ABB RobotStudio station: 501_cocktailBot_v1_20220412-142528.rsstn

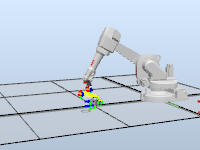
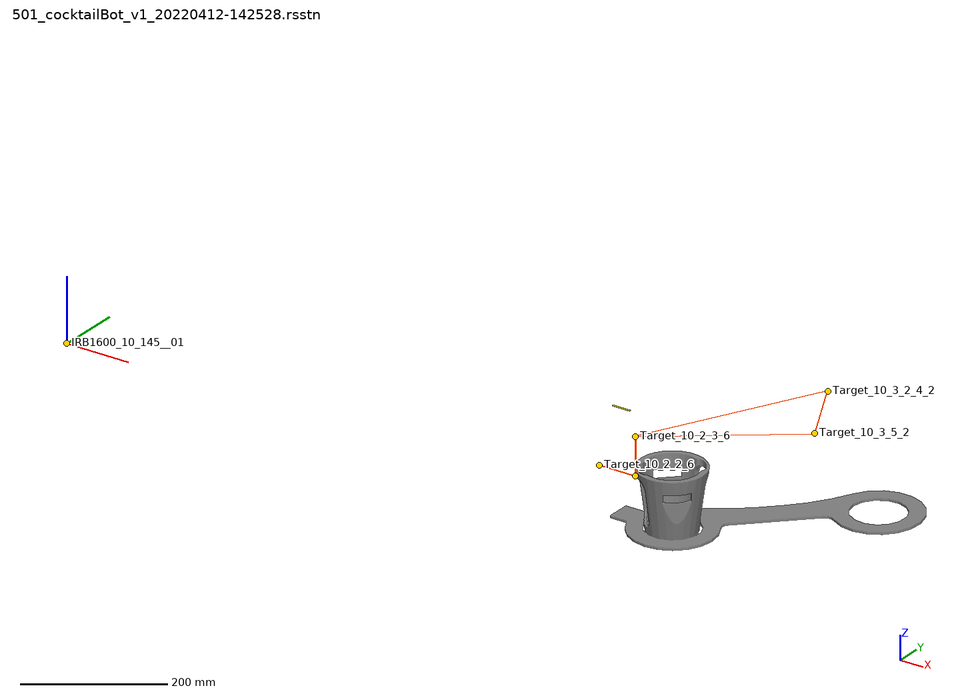
[picture v1: parts stored in the station drawn from their meshes, with robot base, taught points and paths (robot models come from the ABB library and are not in the file)]
Station 501_cocktailBot_v1 (saved by RobotStudio 21.4.9700.0)
Controller IRB1600_10_145
  mechanical unit ROB_1: IRB1600_10_145__01, 6 joints, base frame (0, 0, 0) mm
Layout (positions relative to the parent item):
  - GS25_Gripper [mechanism] at (1000, -191.15, 290.13) mm, rotated rx -130 ry 0 rz 0 deg; joint values [0, 0] (rad or m)
      TCP GS25_Gripper_1 at (0, 0, 90.5) mm
      links: L1, L2, L3
  - Gripper_SC [smart component] at (990, 0, 0) mm, rotated rx 0 ry 90 rz 0 deg
      signals: DI Gripper_Attach, DO Attached
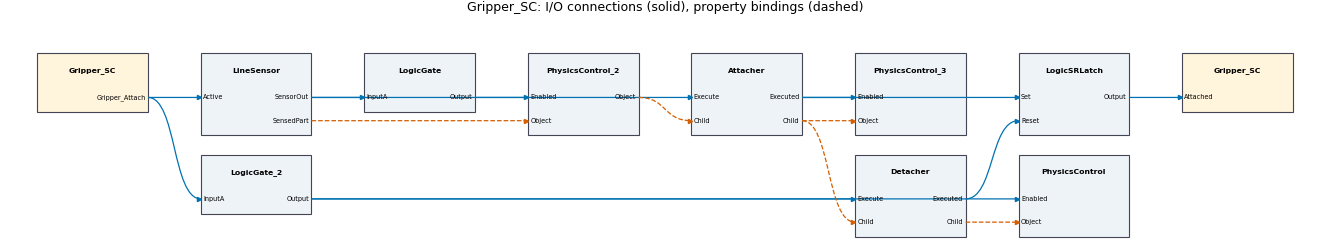
      connections:
        Gripper_SC.Gripper_Attach -> LineSensor.Active
        LineSensor.SensorOut -> LogicGate.InputA
        LogicGate.Output -> PhysicsControl_2.Enabled
        LineSensor.SensorOut -> Attacher.Execute
        Attacher.Executed -> LogicSRLatch.Set
        LogicSRLatch.Output -> Gripper_SC.Attached
        Gripper_SC.Gripper_Attach -> LogicGate_2.InputA
        LogicGate_2.Output -> Detacher.Execute
        Detacher.Executed -> LogicSRLatch.Reset
        LogicGate_2.Output -> PhysicsControl.Enabled
        Attacher.Executed -> PhysicsControl_3.Enabled
        LineSensor.SensedPart => PhysicsControl_2.Object
        PhysicsControl_2.Object => Attacher.Child
        Detacher.Child => PhysicsControl.Object
        Attacher.Child => Detacher.Child
        Attacher.Child => PhysicsControl_3.Object
    - LineSensor [smart component, from Components\LineSensor.rslib] at (-231.47, -121.24, -10.63) mm, rotated rx 0 ry 0 rz 50 deg
        properties: Start=[2.85358248322543E-07 0 0.00610500428453198]; End=[2.85358248322543E-07 0 0.0350726372106779]; Radius=0.001; SensedPart=(none); SensedPoint=[0 0 0]
      - _sensorPart_ [part], size 2 x 2 x 29 mm
    - Attacher [smart component, from Components\Attacher.rslib]
        properties: Parent=GS25_Gripper; Flange=0; Child=cup; Mount=false; Offset=[0 0 0]; Orientation=[0 0 0]
    - Detacher [smart component, from Components\Detacher.rslib]
        properties: Child=cup; KeepPosition=true
    - LogicGate [smart component, from Components\LogicGate.rslib]
        properties: Operator=NOT; Delay=0
    - LogicSRLatch [smart component, from Components\LogicSRLatch.rslib]
    - PhysicsControl [smart component, from Components\PhysicsControl.rslib]
        properties: Object=cup; Behavior=0; SurfaceVelocity=0
    - LogicGate_2 [smart component, from Components\LogicGate.rslib]
        properties: Operator=NOT; Delay=0
    - PhysicsControl_2 [smart component, from Components\PhysicsControl.rslib]
        properties: Object=(none); Behavior=3; SurfaceVelocity=0
  - SmartComponent_1 [smart component] at (1000, -121.83, 231.96) mm, rotated rx -130 ry 0 rz 0 deg
      signals: DI Reset_cube, DI Reset_objects
      connections:
        SmartComponent_1.Reset_objects -> Positioner.Execute
        Positioner.Executed -> Positioner_2.Execute
        Positioner_2.Executed -> Positioner_3.Execute
    - Positioner [smart component, from Components\Positioner.rslib]
        properties: Object=(none); Position=[-0.449454 -0.908727 0]; Orientation=[1.5707963267949 0 1.5707963267949]; Reference=Global; ReferenceObject=(none)
    - Positioner_2 [smart component, from Components\Positioner.rslib]
        properties: Object=(none); Position=[-0.498778 -0.908734 0.000796]; Orientation=[1.5707963267949 0 -1.56573487196411]; Reference=Global; ReferenceObject=(none)
    - Positioner_3 [smart component, from Components\Positioner.rslib]
        properties: Object=(none); Position=[-0.452858 -1.056064 0.000796]; Orientation=[1.5707963267949 0 -1.37980494674916]; Reference=Global; ReferenceObject=(none)
  - Toolside_plates [part] at (0, 0, 0) mm
  - Toolplate2 [part, from Libraries\gs25V2.rslib] at (0, 0, 0) mm
  - cup [part] at (1000, -1.82, 0) mm, rotated rx 90 ry 0 rz 0 deg, size 101.6 x 95 x 100.9 mm
  - cupHolderHolder_3 [part] at (1000, 0, -1.59) mm, rotated rx -90 ry 0 rz 0 deg, size 355.2 x 3.2 x 329.2 mm
  - IRB1600_10_145__01 [mechanism, from Robots\IRB1600_10_145_G_01.rslib] at (0, 0, 0) mm; joint values [-0.2364, 1.0092, 0.0645, 1.0133, 1.0708, 2.1274] (rad or m)
Attachment: LineSensor is attached to GS25_Gripper / L1
Attachment: SmartComponent_1 is attached to GS25_Gripper / L1
Attachment: GS25_Gripper is attached to IRB1600_10_145__01 / Link6
EventTableEntry 1061: Group=, Trigger=DO_Gripper 1062, Actions=[EventTableActionMechanicalPose 1063], Comment=, ActivationMode=2, Cyclic=false
EventTableTriggerIO 1062: IOValue=[1], IRC5Controller=? -1, Operator=0, SignalSource=? -1
EventTableActionMechanicalPose 1063: VirtualSignal=, Mechanism=GS25_Gripper 1072, ToPoseName=Gripper_Open, VirtualSignalValue=[1]
EventTableEntry 1064: Group=, Trigger=DO_Gripper 1065, Actions=[EventTableActionMechanicalPose 1066], Comment=, ActivationMode=2, Cyclic=false
EventTableTriggerIO 1065: IOValue=[0], IRC5Controller=? -1, Operator=0, SignalSource=? -1
EventTableActionMechanicalPose 1066: VirtualSignal=, Mechanism=GS25_Gripper 1072, ToPoseName=Gripper_Closed, VirtualSignalValue=[1]
EventTableTriggerIO 1240: IOValue=[1], IRC5Controller=? -1, Operator=0, SignalSource=? -1
EventTableTriggerIO 1241: IOValue=[0], IRC5Controller=? -1, Operator=0, SignalSource=? -1
EventTableTriggerIO 1347: IOValue=[1], IRC5Controller=? -1, Operator=0, SignalSource=? -1
EventTableTriggerIO 1348: IOValue=[1], IRC5Controller=? -1, Operator=0, SignalSource=? -1
EventTableTriggerIO 1349: IOValue=[1], IRC5Controller=? -1, Operator=0, SignalSource=? -1
EventTableTriggerIO 1350: IOValue=[1], IRC5Controller=? -1, Operator=0, SignalSource=? -1
EventTableTriggerIO 1351: IOValue=[1], IRC5Controller=? -1, Operator=0, SignalSource=? -1
EventTableTriggerIO 1352: IOValue=[1], IRC5Controller=? -1, Operator=0, SignalSource=? -1
EventTableTriggerIO 1353: IOValue=[0], IRC5Controller=? -1, Operator=0, SignalSource=? -1
EventTableTriggerIO 1354: IOValue=[0], IRC5Controller=? -1, Operator=0, SignalSource=? -1
EventTableTriggerIO 1355: IOValue=[0], IRC5Controller=? -1, Operator=0, SignalSource=? -1
EventTableTriggerIO 1356: IOValue=[0], IRC5Controller=? -1, Operator=0, SignalSource=? -1
EventTableTriggerIO 1357: IOValue=[0], IRC5Controller=? -1, Operator=0, SignalSource=? -1
EventTableTriggerIO 1358: IOValue=[0], IRC5Controller=? -1, Operator=0, SignalSource=? -1
EventTableTriggerIO 1359: IOValue=[1], IRC5Controller=? -1, Operator=0, SignalSource=? -1
EventTableTriggerIO 1360: IOValue=[0], IRC5Controller=? -1, Operator=0, SignalSource=? -1
EventTableTriggerIO 2021: IOValue=[1], IRC5Controller=? -1, Operator=0, SignalSource=? -1
EventTableTriggerIO 2022: IOValue=[0], IRC5Controller=? -1, Operator=0, SignalSource=? -1
EventTableTriggerIO 2984: IOValue=[1], IRC5Controller=? -1, Operator=0, SignalSource=? -1
EventTableTriggerIO 2985: IOValue=[1], IRC5Controller=? -1, Operator=0, SignalSource=? -1
EventTableTriggerIO 2986: IOValue=[1], IRC5Controller=? -1, Operator=0, SignalSource=? -1
EventTableTriggerIO 2987: IOValue=[1], IRC5Controller=? -1, Operator=0, SignalSource=? -1
EventTableTriggerIO 2988: IOValue=[1], IRC5Controller=? -1, Operator=0, SignalSource=? -1
EventTableTriggerIO 2989: IOValue=[1], IRC5Controller=? -1, Operator=0, SignalSource=? -1
EventTableTriggerIO 2990: IOValue=[0], IRC5Controller=? -1, Operator=0, SignalSource=? -1
EventTableTriggerIO 2991: IOValue=[0], IRC5Controller=? -1, Operator=0, SignalSource=? -1
EventTableTriggerIO 2992: IOValue=[0], IRC5Controller=? -1, Operator=0, SignalSource=? -1
EventTableTriggerIO 2993: IOValue=[0], IRC5Controller=? -1, Operator=0, SignalSource=? -1
EventTableTriggerIO 2994: IOValue=[0], IRC5Controller=? -1, Operator=0, SignalSource=? -1
EventTableTriggerIO 2995: IOValue=[0], IRC5Controller=? -1, Operator=0, SignalSource=? -1
EventTableTriggerIO 3347: IOValue=[1], IRC5Controller=? -1, Operator=0, SignalSource=? -1
EventTableTriggerIO 3348: IOValue=[0], IRC5Controller=? -1, Operator=0, SignalSource=? -1
EventTableTriggerIO 3367: IOValue=[1], IRC5Controller=? -1, Operator=0, SignalSource=? -1
EventTableTriggerIO 3368: IOValue=[1], IRC5Controller=? -1, Operator=0, SignalSource=? -1
EventTableTriggerIO 3369: IOValue=[1], IRC5Controller=? -1, Operator=0, SignalSource=? -1
EventTableTriggerIO 3370: IOValue=[1], IRC5Controller=? -1, Operator=0, SignalSource=? -1
EventTableTriggerIO 3371: IOValue=[1], IRC5Controller=? -1, Operator=0, SignalSource=? -1
EventTableTriggerIO 3372: IOValue=[1], IRC5Controller=? -1, Operator=0, SignalSource=? -1
EventTableTriggerIO 3373: IOValue=[1], IRC5Controller=? -1, Operator=0, SignalSource=? -1
EventTableTriggerIO 3374: IOValue=[1], IRC5Controller=? -1, Operator=0, SignalSource=? -1
EventTableTriggerIO 3375: IOValue=[1], IRC5Controller=? -1, Operator=0, SignalSource=? -1
EventTableTriggerIO 3376: IOValue=[1], IRC5Controller=? -1, Operator=0, SignalSource=? -1
EventTableTriggerIO 3377: IOValue=[1], IRC5Controller=? -1, Operator=0, SignalSource=? -1
EventTableTriggerIO 3378: IOValue=[0], IRC5Controller=? -1, Operator=0, SignalSource=? -1
EventTableTriggerIO 3379: IOValue=[0], IRC5Controller=? -1, Operator=0, SignalSource=? -1
EventTableTriggerIO 3380: IOValue=[0], IRC5Controller=? -1, Operator=0, SignalSource=? -1
EventTableTriggerIO 3381: IOValue=[0], IRC5Controller=? -1, Operator=0, SignalSource=? -1
EventTableTriggerIO 3382: IOValue=[0], IRC5Controller=? -1, Operator=0, SignalSource=? -1
EventTableTriggerIO 3383: IOValue=[0], IRC5Controller=? -1, Operator=0, SignalSource=? -1
EventTableTriggerIO 3384: IOValue=[0], IRC5Controller=? -1, Operator=0, SignalSource=? -1
EventTableTriggerIO 3385: IOValue=[0], IRC5Controller=? -1, Operator=0, SignalSource=? -1
EventTableTriggerIO 3386: IOValue=[0], IRC5Controller=? -1, Operator=0, SignalSource=? -1
EventTableTriggerIO 3387: IOValue=[0], IRC5Controller=? -1, Operator=0, SignalSource=? -1
EventTableTriggerIO 3388: IOValue=[0], IRC5Controller=? -1, Operator=0, SignalSource=? -1
EventTableTriggerIO 3593: IOValue=[1], IRC5Controller=? -1, Operator=0, SignalSource=? -1
EventTableTriggerIO 3594: IOValue=[1], IRC5Controller=? -1, Operator=0, SignalSource=? -1
EventTableTriggerIO 3595: IOValue=[1], IRC5Controller=? -1, Operator=0, SignalSource=? -1
EventTableTriggerIO 3596: IOValue=[1], IRC5Controller=? -1, Operator=0, SignalSource=? -1
EventTableTriggerIO 3597: IOValue=[0], IRC5Controller=? -1, Operator=0, SignalSource=? -1
EventTableTriggerIO 3598: IOValue=[0], IRC5Controller=? -1, Operator=0, SignalSource=? -1
EventTableTriggerIO 3599: IOValue=[0], IRC5Controller=? -1, Operator=0, SignalSource=? -1
EventTableTriggerIO 3600: IOValue=[0], IRC5Controller=? -1, Operator=0, SignalSource=? -1
EventTableTriggerIO 3620: IOValue=[1], IRC5Controller=? -1, Operator=0, SignalSource=? -1
EventTableTriggerIO 3621: IOValue=[0], IRC5Controller=? -1, Operator=0, SignalSource=? -1
EventTableTriggerIO 3624: IOValue=[1], IRC5Controller=? -1, Operator=0, SignalSource=? -1
EventTableTriggerIO 3625: IOValue=[1], IRC5Controller=? -1, Operator=0, SignalSource=? -1
EventTableTriggerIO 3626: IOValue=[1], IRC5Controller=? -1, Operator=0, SignalSource=? -1
EventTableTriggerIO 3627: IOValue=[0], IRC5Controller=? -1, Operator=0, SignalSource=? -1
EventTableTriggerIO 3628: IOValue=[0], IRC5Controller=? -1, Operator=0, SignalSource=? -1
EventTableTriggerIO 3629: IOValue=[0], IRC5Controller=? -1, Operator=0, SignalSource=? -1
EventTableTriggerIO 3630: IOValue=[1], IRC5Controller=? -1, Operator=0, SignalSource=? -1
EventTableTriggerIO 3631: IOValue=[0], IRC5Controller=? -1, Operator=0, SignalSource=? -1
EventTableTriggerIO 4343: IOValue=[1], IRC5Controller=? -1, Operator=0, SignalSource=? -1
EventTableTriggerIO 4344: IOValue=[0], IRC5Controller=? -1, Operator=0, SignalSource=? -1
Station logic (signal -> signal, property => property):
  IRB_1600_8kg_1.45m.DO_Attach_me -> Gripper_SC.Gripper_Attach
  IRB_1600_8kg_1.45m.DO_Reset_blocks -> SmartComponent_1.Reset_objects
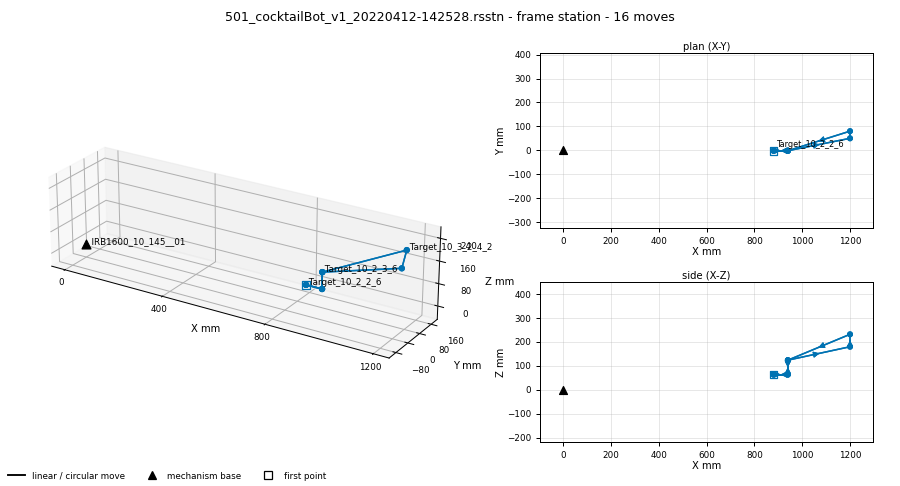
[picture p0: tool path of 501_cocktailBot_v1_20220412-142528.rsstn in frame station, 16 of 17 moves have a stored position in this frame; points joined in program order, loops and branches not executed]
Targets, tools, work objects and paths stored in the station, written as RAPID:
! task (no controller)
MODULE CalibData
  PERS tooldata GS25_Gripper_TCP:=[TRUE,[[0,0,140],[0.991444861,0,0,-0.130526192]],[1,[1,1,1],[1,0,0,0],0,0,0]];
  PERS tooldata Toolside_plate_TCP:=[TRUE,[[0,0,110],[1,0,0,0]],[1,[0,0,7.9375],[1,0,0,0],0,0,0]];
  PERS wobjdata Target_10:=[FALSE,TRUE,"",[[1000,-1.825,0],[1,0,0,0]],[[0,0,0],[1,0,0,0]]];
  PERS wobjdata Workobject_2:=[FALSE,TRUE,"",[[909.454,-18.777,3.412],[1,0,0,0]],[[0,0,0],[1,0,0,0]]];
  PERS wobjdata Target_20:=[FALSE,TRUE,"",[[1200,200,0.237],[1,0,0,0]],[[0,0,0],[1,0,0,0]]];
ENDMODULE

! task (no controller)
MODULE Module1
  CONST robtarget Target_10_2:=[[-60,0,64],[0.5,-0.5,0.5,-0.5],[0,0,0,0],[9E+09,9E+09,9E+09,9E+09,9E+09,9E+09]];
  CONST robtarget Target_10_3:=[[0,-150,180],[0.707106781,-0.707106781,0,0],[0,0,0,0],[9E+09,9E+09,9E+09,9E+09,9E+09,9E+09]];
  CONST robtarget Target_10_2_2:=[[-120,0,64],[0.5,-0.5,0.5,-0.5],[0,0,0,0],[9E+09,9E+09,9E+09,9E+09,9E+09,9E+09]];
  CONST robtarget Target_10_2_3:=[[-60,0,124],[0.5,-0.5,0.5,-0.5],[0,0,0,0],[9E+09,9E+09,9E+09,9E+09,9E+09,9E+09]];
  CONST robtarget Target_10_3_2:=[[0,-120.00000003,231.961524244],[0.422618262,-0.906307787,0,0],[0,0,0,0],[9E+09,9E+09,9E+09,9E+09,9E+09,9E+09]];
  CONST robtarget Target_10_2_6:=[[-60,0,64],[0.5,-0.5,0.5,-0.5],[0,0,0,0],[9E+09,9E+09,9E+09,9E+09,9E+09,9E+09]];
  CONST robtarget Target_10_2_2_4:=[[-120,0,64],[0.5,-0.5,0.5,-0.5],[0,0,0,0],[9E+09,9E+09,9E+09,9E+09,9E+09,9E+09]];
  CONST robtarget Target_10_2_3_4:=[[-60,0,124],[0.5,-0.5,0.5,-0.5],[0,0,0,0],[9E+09,9E+09,9E+09,9E+09,9E+09,9E+09]];
  CONST robtarget Target_10_3_5:=[[0,-150,180],[0.707106781,-0.707106781,0,0],[0,0,0,0],[9E+09,9E+09,9E+09,9E+09,9E+09,9E+09]];
  CONST robtarget Target_10_3_2_4:=[[0,-120.00000003,231.961524244],[0.422618262,-0.906307787,0,0],[0,0,0,0],[9E+09,9E+09,9E+09,9E+09,9E+09,9E+09]];
  CONST robtarget Target_10_2_8:=[[30.546,16.952,60.588],[0.5,-0.5,0.5,-0.5],[0,0,0,0],[9E+09,9E+09,9E+09,9E+09,9E+09,9E+09]];
  CONST robtarget Target_10_2_2_6:=[[-29.454,16.952,60.588],[0.5,-0.5,0.5,-0.5],[0,0,0,0],[9E+09,9E+09,9E+09,9E+09,9E+09,9E+09]];
  CONST robtarget Target_10_2_3_6:=[[30.546,16.952,120.588],[0.5,-0.5,0.5,-0.5],[0,0,0,0],[9E+09,9E+09,9E+09,9E+09,9E+09,9E+09]];
  CONST robtarget Target_10_3_7:=[[90.546,-133.048,176.588],[0.707106781,-0.707106781,0,0],[0,0,0,0],[9E+09,9E+09,9E+09,9E+09,9E+09,9E+09]];
  CONST robtarget Target_10_3_2_6:=[[90.546,-103.04800003,228.549524244],[0.422618262,-0.906307787,0,0],[0,0,0,0],[9E+09,9E+09,9E+09,9E+09,9E+09,9E+09]];
  CONST robtarget Target_10_2_2_4_2:=[[170.546,218.777,60.825],[0.5,-0.5,0.5,-0.5],[0,0,0,0],[9E+09,9E+09,9E+09,9E+09,9E+09,9E+09]];
  CONST robtarget Target_10_2_3_4_2:=[[230.546,218.777,120.825],[0.5,-0.5,0.5,-0.5],[0,0,0,0],[9E+09,9E+09,9E+09,9E+09,9E+09,9E+09]];
  CONST robtarget Target_10_2_6_2:=[[230.546,218.777,60.825],[0.5,-0.5,0.5,-0.5],[0,0,0,0],[9E+09,9E+09,9E+09,9E+09,9E+09,9E+09]];
  CONST robtarget Target_10_3_2_4_2:=[[290.546,98.77699997,228.786524244],[0.422618262,-0.906307787,0,0],[0,0,0,0],[9E+09,9E+09,9E+09,9E+09,9E+09,9E+09]];
  CONST robtarget Target_10_3_5_2:=[[290.546,68.777,176.825],[0.707106781,-0.707106781,0,0],[0,0,0,0],[9E+09,9E+09,9E+09,9E+09,9E+09,9E+09]];
  PROC Path_10()
    MoveL Target_10_2_2_6,v1000,z100,GS25_Gripper_TCP\WObj:=Workobject_2;
    MoveL Target_10_2_8,v1000,z100,GS25_Gripper_TCP\WObj:=Workobject_2;
    MoveL Target_10_2_3_6,v1000,z100,GS25_Gripper_TCP\WObj:=Workobject_2;
    MoveL Target_10_3_5_2,v1000,z100,GS25_Gripper_TCP\WObj:=Workobject_2;
    MoveL Target_10_3_2_4_2,v1000,z100,GS25_Gripper_TCP\WObj:=Workobject_2;
    MoveL Target_10_2_3_6,v1000,z100,GS25_Gripper_TCP\WObj:=Workobject_2;
    MoveL Target_10_2_8,v1000,z100,GS25_Gripper_TCP\WObj:=Workobject_2;
    MoveL Target_10_2_2_6,v1000,z100,GS25_Gripper_TCP\WObj:=Workobject_2;
  ENDPROC
  PROC Path_20()
  ENDPROC
ENDMODULE

! task T_ROB1
MODULE Module1
  CONST jointtarget jt_Home:=[[0,0,0,0,0,0],[9E+09,9E+09,9E+09,9E+09,9E+09,9E+09]];
  CONST robtarget Target_10_2_8:=[[30.546,16.952,60.588],[0.5,-0.5,0.5,-0.5],[0,0,0,0],[9E+09,9E+09,9E+09,9E+09,9E+09,9E+09]];
  CONST robtarget Target_10_2_2_6:=[[-29.454,16.952,60.588],[0.5,-0.5,0.5,-0.5],[0,0,0,0],[9E+09,9E+09,9E+09,9E+09,9E+09,9E+09]];
  CONST robtarget Target_10_2_3_6:=[[30.546,16.952,120.588],[0.5,-0.5,0.5,-0.5],[0,0,0,0],[9E+09,9E+09,9E+09,9E+09,9E+09,9E+09]];
  CONST robtarget Target_10_3_7:=[[90.546,-133.048,176.588],[0.707106781,-0.707106781,0,0],[0,0,0,0],[9E+09,9E+09,9E+09,9E+09,9E+09,9E+09]];
  CONST robtarget Target_10_3_2_6:=[[90.546,-103.04800003,228.549524244],[0.422618262,-0.906307787,0,0],[0,0,0,0],[9E+09,9E+09,9E+09,9E+09,9E+09,9E+09]];
  CONST robtarget Target_10_2_2_4_2:=[[170.546,218.777,60.825],[0.5,-0.5,0.5,-0.5],[0,0,0,0],[9E+09,9E+09,9E+09,9E+09,9E+09,9E+09]];
  CONST robtarget Target_10_2_3_4_2:=[[230.546,218.777,120.825],[0.5,-0.5,0.5,-0.5],[0,0,0,0],[9E+09,9E+09,9E+09,9E+09,9E+09,9E+09]];
  CONST robtarget Target_10_2_6_2:=[[230.546,218.777,60.825],[0.5,-0.5,0.5,-0.5],[0,0,0,0],[9E+09,9E+09,9E+09,9E+09,9E+09,9E+09]];
  CONST robtarget Target_10_3_2_4_2:=[[290.546,98.77699997,228.786524244],[0.422618262,-0.906307787,0,0],[0,0,0,0],[9E+09,9E+09,9E+09,9E+09,9E+09,9E+09]];
  CONST robtarget Target_10_3_5_2:=[[290.546,68.777,176.825],[0.707106781,-0.707106781,0,0],[0,0,0,0],[9E+09,9E+09,9E+09,9E+09,9E+09,9E+09]];
ENDMODULE

! task T_ROB1
MODULE MainModule
  CONST jointtarget home:=[[0,0,0,0,0,0],[0,0,0,0,0,0]];
  PROC main()
    MoveAbsJ home,v1000,fine,tool0;
  ENDPROC
ENDMODULE

! task T_ROB1
MODULE CalibData
  PERS tooldata GS25_Gripper_TCP:=[TRUE,[[0,0,140],[0.991444861,0,0,-0.130526192]],[1,[1,1,1],[1,0,0,0],0,0,0]];
  PERS wobjdata Workobject_2:=[FALSE,TRUE,"",[[1010.502772549,-872.780780396,3.412],[0.999963549,0,0,-0.008538136]],[[0,0,0],[1,0,0,0]]];
ENDMODULE

! task T_ROB1
MODULE CalibData
  PERS tooldata GS25_Gripper_TCP:=[TRUE,[[1324.163842548,0,-166.519052838],[0.5,0,-0.866025404,0]],[1,[1,1,1],[1,0,0,0],0,0,0]];
  PERS wobjdata Workobject_2:=[FALSE,TRUE,"",[[909.454,-18.777,3.412],[1,0,0,0]],[[0,0,0],[1,0,0,0]]];
  PERS tooldata GS25_Gripper_1:=[TRUE,[[0,0,90.5],[1,0,0,0]],[1,[1,1,1],[1,0,0,0],0,0,0]];
ENDMODULE

! task T_ROB1
MODULE Module1
  CONST robtarget Target_10_2_8:=[[30.546,16.952,60.588],[0.5,-0.5,0.5,-0.5],[0,0,0,0],[9E+09,9E+09,9E+09,9E+09,9E+09,9E+09]];
  CONST robtarget Target_10_2_2_6:=[[-29.454,16.952,60.588],[0.5,-0.5,0.5,-0.5],[0,0,0,0],[9E+09,9E+09,9E+09,9E+09,9E+09,9E+09]];
  CONST robtarget Target_10_2_3_6:=[[30.546,16.952,120.588],[0.5,-0.5,0.5,-0.5],[0,0,0,0],[9E+09,9E+09,9E+09,9E+09,9E+09,9E+09]];
  CONST robtarget Target_10_3_7:=[[90.546,-133.048,176.588],[0.707106781,-0.707106781,0,0],[0,0,0,0],[9E+09,9E+09,9E+09,9E+09,9E+09,9E+09]];
  CONST robtarget Target_10_3_2_6:=[[90.546,-103.04800003,228.549524244],[0.422618262,-0.906307787,0,0],[0,0,0,0],[9E+09,9E+09,9E+09,9E+09,9E+09,9E+09]];
  CONST robtarget Target_10_2_2_4_2:=[[170.546,218.777,60.825],[0.5,-0.5,0.5,-0.5],[0,0,0,0],[9E+09,9E+09,9E+09,9E+09,9E+09,9E+09]];
  CONST robtarget Target_10_2_3_4_2:=[[230.546,218.777,120.825],[0.5,-0.5,0.5,-0.5],[0,0,0,0],[9E+09,9E+09,9E+09,9E+09,9E+09,9E+09]];
  CONST robtarget Target_10_2_6_2:=[[230.546,218.777,60.825],[0.5,-0.5,0.5,-0.5],[0,0,0,0],[9E+09,9E+09,9E+09,9E+09,9E+09,9E+09]];
  CONST robtarget Target_10_3_2_4_2:=[[290.546,98.77699997,228.786524244],[0.422618262,-0.906307787,0,0],[0,0,0,0],[9E+09,9E+09,9E+09,9E+09,9E+09,9E+09]];
  CONST robtarget Target_10_3_5_2:=[[290.546,68.777,176.825],[0.707106781,-0.707106781,0,0],[0,0,0,0],[9E+09,9E+09,9E+09,9E+09,9E+09,9E+09]];
  CONST robtarget Target_10_2_2_6_2:=[[-29.454,16.952,60.588],[0.5,-0.5,0.5,-0.5],[0,0,0,0],[9E+09,9E+09,9E+09,9E+09,9E+09,9E+09]];
  CONST robtarget Target_10_2_8_2:=[[30.546,16.952,60.588],[0.5,-0.5,0.5,-0.5],[0,0,0,0],[9E+09,9E+09,9E+09,9E+09,9E+09,9E+09]];
  CONST robtarget Target_10_2_3_6_3:=[[30.546,16.952,120.588],[0.5,-0.5,0.5,-0.5],[0,0,0,0],[9E+09,9E+09,9E+09,9E+09,9E+09,9E+09]];
  CONST robtarget Target_10_3_5_2_2:=[[290.546,68.777,176.825],[0.707106781,-0.707106781,0,0],[0,0,0,0],[9E+09,9E+09,9E+09,9E+09,9E+09,9E+09]];
  CONST robtarget Target_10_3_2_4_2_2:=[[290.546,98.77699997,228.786524244],[0.422618262,-0.906307787,0,0],[0,0,0,0],[9E+09,9E+09,9E+09,9E+09,9E+09,9E+09]];
  PROC Path_10()
    MoveJ Target_10_2_2_6_2,v1000,z100,GS25_Gripper_TCP\WObj:=Workobject_2;
    MoveL Target_10_2_8_2,v1000,z100,GS25_Gripper_TCP\WObj:=Workobject_2;
    MoveL Target_10_2_3_6_3,v1000,z100,GS25_Gripper_TCP\WObj:=Workobject_2;
    MoveL Target_10_3_5_2_2,v1000,z100,GS25_Gripper_TCP\WObj:=Workobject_2;
    MoveL Target_10_3_2_4_2_2,v1000,z100,GS25_Gripper_TCP\WObj:=Workobject_2;
    MoveL Target_10_2_3_6_3,v1000,z100,GS25_Gripper_TCP\WObj:=Workobject_2;
    MoveL Target_10_2_8_2,v1000,z100,GS25_Gripper_TCP\WObj:=Workobject_2;
    MoveL Target_10_2_2_6_2,v1000,z100,GS25_Gripper_TCP\WObj:=Workobject_2;
  ENDPROC
  PROC main()
    Path_10;
  ENDPROC
ENDMODULE

